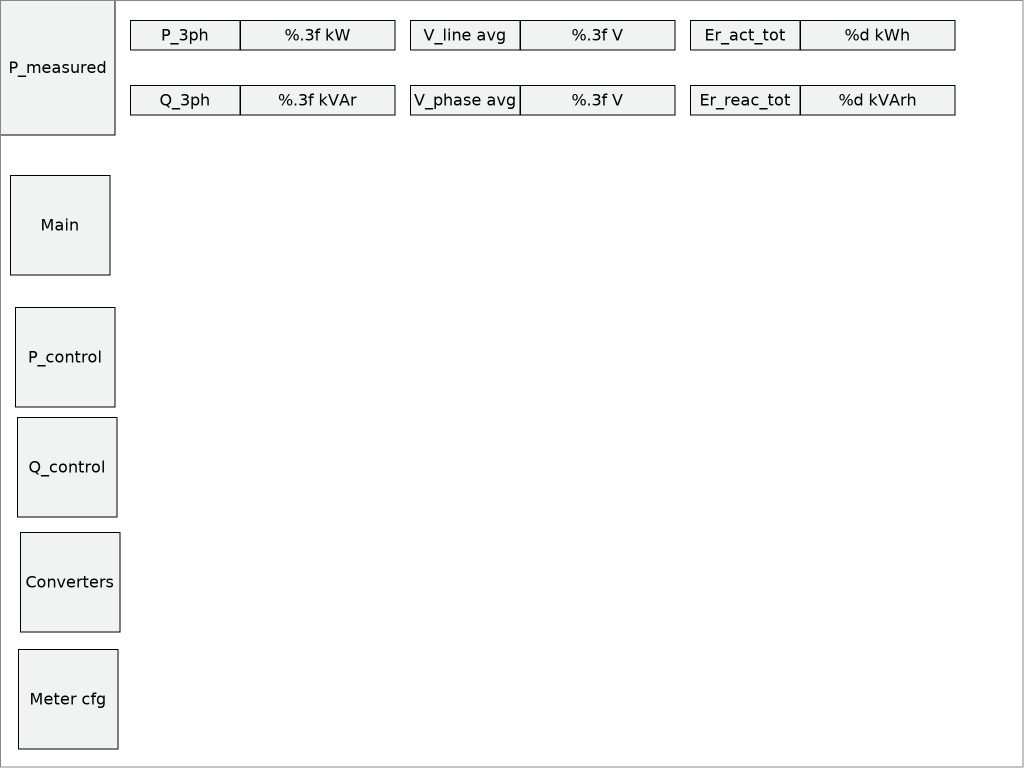
VISUALIZATION Main_GUI  // 1024x768
    Rectangle (130,20 110x30), "P_3ph"
    Rectangle (0,0 115x135), "P_measured"
    Rectangle (240,20 155x30), "%.3f kW", text variable: GVL_POWERMETER.Power_analyzer.P_kW
    Rectangle (130,85 110x30), "Q_3ph"
    Rectangle (240,85 155x30), "%.3f kVAr", text variable: GVL_POWERMETER.Power_analyzer.Q_kVAr
    Rectangle (410,20 110x30), "V_line avg"
    Rectangle (520,20 155x30), "%.3f V", text variable: GVL_POWERMETER.V_line_avg_Volt
    Rectangle (410,85 110x30), "V_phase avg"
    Rectangle (520,85 155x30), "%.3f V", text variable: GVL_POWERMETER.V_phase_avg_pu
    Rectangle (690,20 110x30), "Er_act_tot"
    Rectangle (800,20 155x30), "%d kWh", text variable: GVL_POWERMETER.Active_er_tot_kWh
    Rectangle (690,85 110x30), "Er_reac_tot"
    Rectangle (800,85 155x30), "%d kVArh", text variable: GVL_POWERMETER.React_er_tot_kVArh
    Rectangle (10,175 100x100), "Main"
    Rectangle (15,307 100x100), "P_control"
    Rectangle (17,417 100x100), "Q_control"
    Rectangle (18,649 100x100), "Meter cfg"
    Rectangle (20,532 100x100), "Converters"
END_VISUALIZATION

(* stored: Version 1.1.0.1, ProductVersion 3.1.4024.11
   Visu Main_GUI: Id {7bd4137f-6365-4ffe-add0-0c67551971ac} *)
